(* CoDeSys 2.3.9.41 project: AVO_M.pro *)
(* Libraries: STANDARD.LIB 4.10.05 11:14:46, IECSFC.LIB 13.4.06 15:51:28, SYSLIBTIME.LIB 20.2.06 13:31:16, SYSTASKINFO.LIB 20.2.06 13:31:38, ANALYZATION.LIB 5.10.99 09:05:06, SYSLIBCALLBACK.LIB 20.2.06 13:31:08, Util.lib 18.5.10 15:14:28 *)

(* PLC configuration (modules and I/O channels)
Fast discrete inputs [I_SIMPLE_INPUT] node 0, in %IB0 out %QB0 {Filtrationtime = 10}
  AT %IX0.0 [BitInput] Discrete input 1
  AT %IX0.1 [BitInput] Discrete input 2
  AT %IX0.2 [BitInput] Discrete input 3
  AT %IX0.3 [BitInput] Discrete input 4
Discrete inputs [ID130] node 1, in %IB1 out %QB1 {Filtrationtime_GeneralINP = 10; Visibility = No; PinCount = 12}
  AT %IB1.0 [ByteInput] 8 discrete inputs
  AT %IB1.1 [ByteInput] 4 discrete inputs
Discrete outputs [ID131] node 2, in %IB2 out %QB2 {SafeValueByte = 0; SafeValueByteM = 0; Visibility = No; PinCount = 12}
  AT %QB2.0 [ByteOutput] 8 discrete outputs
  AT %QB2.1 [ByteOutput] 4 discrete outputs
Fast analog inputs [ID125] node 3, in %IB3 out %QB3 {Flt_Comm = 50Hz 2Por}
  AT %IR3.0 [FloatInputP] AI #1 {AIN_TYPE = 4-20 mA; Peak_Filtr = 200; Flt_Ch = Avr 4; TauRC = 10; MinFV = -50; MaxFV = 150}
  AT %IR3.1 [FloatInputP] AI #2 {AIN_TYPE = 4-20 mA; Peak_Filtr = 200; Flt_Ch = Off; TauRC = 10; MinFV = -50; MaxFV = 150}
  AT %IR3.2 [FloatInputP] AI #3 {AIN_TYPE = 4-20 mA; Peak_Filtr = 200; Flt_Ch = Off; TauRC = 10; MinFV = -50; MaxFV = 150}
  AT %IR3.3 [FloatInputP] AI #4 {AIN_TYPE = 4-20 mA; Peak_Filtr = 200; Flt_Ch = Off; TauRC = 10; MinFV = -50; MaxFV = 150}
  AT %IR3.4 [FloatInputP] AI #5 {AIN_TYPE = 4-20 mA; Peak_Filtr = 200; Flt_Ch = Off; TauRC = 10; MinFV = 0; MaxFV = 1.6}
  AT %IR3.5 [FloatInputP] AI #6 {AIN_TYPE = 4-20 mA; Peak_Filtr = 200; Flt_Ch = Off; TauRC = 10; MinFV = 0; MaxFV = 1.6}
  AT %IR3.6 [FloatInputP] AI #7 {AIN_TYPE = 4-20 mA; Peak_Filtr = 200; Flt_Ch = Off; TauRC = 10; MinFV = 0; MaxFV = 20000.0}
  AT %IR3.7 [FloatInputP] AI #8 {AIN_TYPE = 4-20 mA; Peak_Filtr = 200; Flt_Ch = Off; TauRC = 10; MinFV = 0; MaxFV = 20000.0}
  AT %IW3.8 [WordInput] AI read time (10ms)
Analog outputs [ID126] node 4, in %IB4 out %QB4
  AT %QR4.0 [FloatOutputP] AO #1 {AOUT_TYPE = 0-10V; SafeValueREAL = 0.0}
  AT %QR4.1 [FloatOutputP] AO #2 {AOUT_TYPE = 0-10V; SafeValueREAL = 0.0}
  AT %QR4.2 [FloatOutputP] AO #3 {AOUT_TYPE = 4-20 mA; SafeValueREAL = 0.0}
  AT %QR4.3 [FloatOutputP] AO #4 {AOUT_TYPE = 4-20 mA; SafeValueREAL = 0.0}
Special input [ID103] node 5, in %IB5 out %QB5 {Filtrationtime = 1000; PinCount = 1; WatchDogPeriod = 400; PollPeriod = 3000; Visibility = No}
  AT %IX5.0 [BitInput] Special input
Special output [ID104] node 6, in %IB6 out %QB6 {Visibility = No; PinCount = 1}
  AT %QX6.0 [BitOutput] Special output
Modbus [MODBUS_ID302] node 0, in %IB7.0 out %QB7.0
  RS-232 [COM2_USART] node 0, in %IB7.0.0 out %QB7.0.0 {CommunicationSpeed = 19200; Parity = EVEN; BitLength = 8 bits; StopLength = One stop bit; InterfaceType = RS232; FrameOriented = RTU; Timeout = 0; Visibility = No}
AT %QB7.1.0 [ByteOutput]
AT %QB7.2.0 [ByteOutput]
AT %QB7.3.0 [ByteOutput]
Float [Float] node 4, in %IB7.4 out %QB7.4
  AT %QD7.4.0 [FloatOutput]
2 byte [Register] node 5, in %IB7.5 out %QB7.5
  AT %QW7.5.0 [WordOutput]
Float [Float] node 6, in %IB7.6 out %QB7.6
  AT %QD7.6.0 [FloatOutput]
Float [Float] node 7, in %IB7.7 out %QB7.7
  AT %QD7.7.0 [FloatOutput]
Float [Float] node 8, in %IB7.8 out %QB7.8
  AT %QD7.8.0 [FloatOutput]
Float [Float] node 9, in %IB7.9 out %QB7.9
  AT %QD7.9.0 [FloatOutput]
Float [Float] node 10, in %IB7.10 out %QB7.10
  AT %QD7.10.0 [FloatOutput]
Float [Float] node 11, in %IB7.11 out %QB7.11
  AT %QD7.11.0 [FloatOutput]
Float [Float] node 12, in %IB7.12 out %QB7.12
  AT %QD7.12.0 [FloatOutput]
  AT %QD7.13.0 [FloatOutput]
Float [Float] node 14, in %IB7.14 out %QB7.14
  AT %QD7.14.0 [FloatOutput]
Float [Float] node 15, in %IB7.15 out %QB7.15
  AT %QD7.15.0 [FloatOutput]
Float [Float] node 16, in %IB7.16 out %QB7.16
  AT %QD7.16.0 [FloatOutput]
  AT %QD7.17.0 [FloatOutput]
RS-485-1 [COM1_USART] node 0, in %IB8.0.0 out %QB8.0.0 {CommunicationSpeed = 9600; Parity = NO PARITY CHECK; BitLength = 8 bits; StopLength = One stop bit; InterfaceType = RS485; FrameOriented = RTU; Timeout = 0; Visibility = No}
8 bits [8Bit] node 1, in %IB8.1 out %QB8.1
  AT %QB8.1.0 [ByteOutput]
8 bits [8Bit] node 2, in %IB8.2 out %QB8.2
  AT %QB8.2.0 [ByteOutput]
8 bits [8Bit] node 3, in %IB8.3 out %QB8.3
  AT %QB8.3.0 [ByteOutput]
8 bits [8Bit] node 4, in %IB8.4 out %QB8.4
  AT %QB8.4.0 [ByteOutput]
8 bits [8Bit] node 5, in %IB8.5 out %QB8.5
  AT %QB8.5.0 [ByteOutput]
8 bits [8Bit] node 6, in %IB8.6 out %QB8.6
  AT %QB8.6.0 [ByteOutput]
8 bits [8Bit] node 7, in %IB8.7 out %QB8.7
  AT %QB8.7.0 [ByteOutput]
8 bits [8Bit] node 8, in %IB8.8 out %QB8.8
  AT %QB8.8.0 [ByteOutput]
8 bits [8Bit] node 9, in %IB8.9 out %QB8.9
  AT %QB8.9.0 [ByteOutput]
8 bits [8Bit] node 10, in %IB8.10 out %QB8.10
  AT %QB8.10.0 [ByteOutput]
8 bits [8Bit] node 11, in %IB8.11 out %QB8.11
  AT %QB8.11.0 [ByteOutput]
  AT %QB8.12.0 [ByteOutput]
8 bits [8Bit] node 13, in %IB8.13 out %QB8.13
  AT %QB8.13.0 [ByteOutput]
8 bits [8Bit] node 14, in %IB8.14 out %QB8.14
  AT %QB8.14.0 [ByteOutput]
8 bits [8Bit] node 15, in %IB8.15 out %QB8.15
  AT %QB8.15.0 [ByteOutput]
8 bits [8Bit] node 16, in %IB8.16 out %QB8.16
  AT %QB8.16.0 [ByteOutput]
8 bits [8Bit] node 17, in %IB8.17 out %QB8.17
  AT %QB8.17.0 [ByteOutput]
8 bits [8Bit] node 18, in %IB8.18 out %QB8.18
  AT %QB8.18.0 [ByteOutput]
8 bits [8Bit] node 19, in %IB8.19 out %QB8.19
  AT %QB8.19.0 [ByteOutput]
8 bits [8Bit] node 20, in %IB8.20 out %QB8.20
  AT %QB8.20.0 [ByteOutput]
*)

(* Global variable list: Global_Variables *)
VAR_GLOBAL RETAIN
(*уставки*)
	Tnorm AT %QD7.6.0:REAL:=15;
	Tust AT %QD7.7.0:REAL:=38;
	Tmax AT %QD7.8.0:REAL:=60;
	Ti AT %QD7.12.0:REAL:=40;
	Kp AT %QD7.13.0:REAL:=0.4;
	tau_vent AT %QW7.5.0:WORD:=10;(*от 300 до 500с*)
END_VAR

VAR_GLOBAL
(*аналоговые входы*)
	t_sec AT %IR3.0:REAL;
	t_in AT %IR3.1:REAL;
	t_out AT %IR3.2:REAL;
	t_air AT %IR3.3:REAL;
	p_in AT %IR3.4:REAL;
	p_out AT %IR3.5:REAL;

(*аналоговые выходы*)
	vent1 AT %QR4.0:REAL:=0;
	vent2 AT %QR4.1:REAL:=0;

(*дискретные входы*)
	vent_kf_overheat AT %IX1.0.0:BOOL:=0; (*0 - авария, 1 - норм*)
	ten_overheat AT %IX1.0.1:BOOL:=0; (*0 - авария, 1 - норм*)
	vent1_crash AT %IX1.0.3:BOOL:=0; (*0 - авария, 1 - норм*)
	vent2_crash AT %IX1.0.4:BOOL:=0; (*0 - авария, 1 - норм*)

	qf1 AT %IX1.0.5:BOOL:=1;
	qf2 AT %IX1.0.6:BOOL:=1;
	qf5 AT %IX1.0.7:BOOL:=1;

(*дискретне выходы*)
	vent_kf AT %QX2.0.0:BOOL:=0;
	ten AT %QX2.0.1:BOOL:=0;

	t_out_high:BOOL:=0; (*превышение Тмакс*)
	p_in_high:BOOL:=0;(*превышение p_in 1,0 МПа*)
	ready:BOOL:=1;
	err:BOOL:=0;

	err_do AT %QX2.0.2:BOOL:=1; (*общая неисправность*)
	ohlad_do AT %QX2.0.3:BOOL:=1;
	norma_do AT %QX2.0.4:BOOL:=1;
	t_out_high_do AT %QX2.0.5:BOOL:=1;
	nagrev_do AT %QX2.0.6:BOOL:=1;
	ready_do AT %QX2.0.7:BOOL:=1;

(*переменные для панели*)
	nagrev AT %QX7.3.0.0:BOOL:=0;(*0-выкл,1-вкл*)
	ohlad AT %QX7.3.0.1:BOOL:=0;(*0-выкл,1-вкл*)
	norma AT %QX7.3.0.2:BOOL:=0;(*0-не норма,1-норма*)
	reg_manu AT %QX7.3.0.3:BOOL:=0;(*0-выкл,1-вкл*)

	vent1_vkl AT %QX7.2.0.0:BOOL:=TRUE;(*0-выкл,1-вкл*)
	vent2_vkl AT %QX7.2.0.1:BOOL:=TRUE;(*0-выкл,1-вкл*)

	Nust AT %QD7.11.0:REAL:=0;(*задание*)

	t_sec_pan AT %QD7.4.0:REAL;
	t_in_pan AT %QD7.9.0:REAL;
	t_out_pan AT %QD7.10.0:REAL;
	t_air_pan AT %QD7.14.0:REAL;
	p_in_pan AT %QD7.15.0:REAL;
	p_out_pan AT %QD7.16.0:REAL;

	err_pan AT %QX7.1.0.7:BOOL:=0;
	vent_kf_overheat_pan AT %QX7.1.0.2:BOOL:=0;
	ten_overheat_pan AT %QX7.1.0.3:BOOL:=0;
	t_out_high_pan AT %QX7.1.0.4:BOOL:=0;
	vent1_crash_pan AT %QX7.1.0.5:BOOL:=0;
	vent2_crash_pan AT %QX7.1.0.6:BOOL:=0;
	qf1_pan AT %QX7.2.0.2:BOOL:=1;
	qf2_pan AT %QX7.2.0.3:BOOL:=1;
	qf5_pan AT %QX7.2.0.4:BOOL:=1;


	vent_kf_pan AT %QX7.1.0.0:BOOL:=0;
	ten_pan AT %QX7.1.0.1:BOOL:=0;

(*наверх*)
	Tust_up AT %QB8.1.0:BYTE:=30;
	Tnorm_up AT %QB8.2.0:BYTE:=80;

	inp1 AT %QB8.3.0:BYTE:=15; (*рольставни, их нет на самом деле*)

	Tmax_up AT %QB8.4.0:BYTE:=160;

	inp3 AT %QB8.5.0:BYTE;
	vent_kf_overheat_up AT %QX8.5.0.2:BOOL:=0;
	ten_overheat_up AT %QX8.5.0.4:BOOL:=0;

	inp2 AT %QB8.6.0:BYTE;
	qf1_up AT %QX8.6.0.0:BOOL:=0;
	qf2_up AT %QX8.6.0.1:BOOL:=0;
	qf5_up AT %QX8.6.0.4:BOOL:=0;

	inp5 AT %QB8.7.0:BYTE;(*зарезервирован*)

	inp4 AT %QB8.8.0:BYTE;
	vent1_crash_up AT %QX8.8.0.0:BOOL:=0;
	vent2_crash_up AT %QX8.8.0.1:BOOL:=0;

	out2 AT %QB8.9.0:BYTE;
	vent1_vkl_up AT %QX8.9.0.0:BOOL:=1;(*0-выкл,1-вкл*)
	vent2_vkl_up AT %QX8.9.0.1:BOOL:=1;(*0-выкл,1-вкл*)
	vent_kf_up AT %QX2.0.0:BOOL:=0;
	ten_up AT %QX2.0.1:BOOL:=0;

	out1 AT %QB8.10.0:BYTE;(*команды на рольставни, их нет*)

	out4 AT %QB8.11.0:BYTE;
	err_up AT %QX8.11.0.0:BOOL:=1; (*0 - есть, 1 - нет*)
	ohlad_up AT %QX8.11.0.1:BOOL:=1; (*0 - есть, 1 - нет*)
	norma_up AT %QX8.11.0.2:BOOL:=1; (*0 - норма, 1 - не норма*)
	t_out_high_up AT %QX8.11.0.3:BOOL:=1; (*0 - есть, 1 - нет*)
	nagrev_up AT %QX8.11.0.4:BOOL:=0; (*0 - есть, 1 - нет*)
	ready_up AT %QX8.11.0.5:BOOL:=0; (*0 - есть, 1 - нет*)

	out3 AT %QB8.12.0:BYTE;
	sys_vkl AT %QX8.12.0.7:BOOL:=0;(*система включена, пока не используется*)

	t_out_up AT %QB8.13.0:BYTE:=90;(*по умолчанию 22*)

	out5 AT %QB8.14.0:BYTE:=0; (*номер режима охлаждения итд*)
	reg_manu_up AT %QX8.14.0.4:BOOL:=0;(*0-авт,1 - ручн*)

	t_sec_up AT %QB8.15.0:BYTE:=80;(*по умолчанию 14*)
	t_in_up AT %QB8.16.0:BYTE:=94;(*по умолчанию 25,2*)
	t_air_up AT %QB8.17.0:BYTE:=100;(*по умолчанию 30*)
	Nust_up AT %QB8.18.0:BYTE:=88;(*по умолчанию 35.2*)
	p_out_up AT %QB8.19.0:BYTE:=125;(*по умолчанию 0,001*)
	p_in_up AT %QB8.20.0:BYTE:=250;(*по умолчанию 0,002*)
END_VAR

(* POU PLC_PRG, ST *)
PROGRAM PLC_PRG
VAR
END_VAR
IF t_sec<Tnorm THEN
	nagrev:=TRUE;
ELSIF vent_kf=FALSE THEN
	nagrev:=FALSE;
END_IF

IF t_sec>=Tnorm-10 THEN
	norma:=TRUE;
ELSE
	norma:=FALSE;
END_IF

IF t_out>=Tust AND p_in>=0.2 AND norma THEN
	ohlad:=TRUE;
END_IF

IF p_in<0.2 THEN
	ohlad:=FALSE;
END_IF

IF nagrev THEN
	Tsec();
END_IF

IF ohlad THEN
	Tout();
END_IF

(*ручное регулирование*)
IF reg_manu THEN
	ohlad:=FALSE;
ELSIF NOT ohlad THEN
	Nust:=0;
END_IF

(*сигналы на вентиляторы*)
vent1:=Nust*BOOL_TO_REAL(vent1_vkl)/10;
vent2:=Nust*BOOL_TO_REAL(vent2_vkl)/10;

(*ошибки*)
errors();

(*передача параметров на панель и на САУ*)
pan();
upperlvl();
END_PROGRAM

(* POU Tsec, ST *)
PROGRAM Tsec
VAR
	delay:TOF;
	tmr:BOOL:=TRUE;
	t: TIME := T#5s;
END_VAR
t:=WORD_TO_TIME(tau_vent*1000);
IF t_sec<Tnorm-5 THEN
	vent_kf:=TRUE;
	ten:=TRUE AND NOT vent_kf_overheat;
	tmr:=TRUE;
END_IF;
IF t_sec>=Tnorm THEN
	delay(IN:=tmr,PT:=t);
	ten:=FALSE;
	tmr:=FALSE;
	vent_kf:=delay.Q;
END_IF;
END_PROGRAM

(* POU Tout, ST *)
PROGRAM Tout
VAR
	reg:PID;
	Td:REAL:=0;
END_VAR
reg(
	ACTUAL:=  t_out,
	SET_POINT:= Tust,
	KP:= -Kp,
	TN:= Ti,
	TV:= Td,
	Y_MANUAL:= Nust,
	Y_OFFSET:= 0,
	Y_MIN:= 0,
	Y_MAX:= 100,
	MANUAL:= reg_manu,
	RESET:= ,
	Y=> Nust,
	LIMITS_ACTIVE=> , 
	OVERFLOW=> );
END_PROGRAM

(* POU errors, ST *)
PROGRAM errors
VAR
END_VAR
t_out_high:=t_out>Tmax;
p_in_high:=p_in>1;

err:=NOT vent_kf_overheat OR NOT  ten_overheat OR NOT vent1_crash OR NOT vent2_crash OR t_out_high OR p_in_high OR NOT qf1 OR NOT qf2 OR NOT qf5;
ready:=NOT err;

IF NOT vent_kf_overheat THEN
ten:=FALSE;
END_IF

IF NOT vent1_crash THEN
vent1_vkl:=FALSE;
END_IF

IF NOT vent2_crash THEN
vent2_vkl:=FALSE;
END_IF
END_PROGRAM

(* POU pan, ST *)
PROGRAM pan
VAR
END_VAR
t_sec_pan:=t_sec;
t_in_pan:=t_in;
t_out_pan:=t_out;
t_air_pan:=t_air;
p_in_pan:=p_in;
p_out_pan:=p_out;

vent_kf_overheat_pan:=vent_kf_overheat;
ten_overheat_pan:=ten_overheat;
t_out_high_pan:=t_out_high;
vent1_crash_pan:=vent1_crash;
vent2_crash_pan:=vent2_crash;

vent_kf_pan:=vent_kf;
ten_pan:=ten;
END_PROGRAM

(* POU upperlvl, ST *)
PROGRAM upperlvl
VAR
END_VAR
Tnorm_up:=REAL_TO_BYTE(Tnorm*2);
Tust_up:=REAL_TO_BYTE(Tust*2);
Tmax_up:=REAL_TO_BYTE(Tmax*2);

(*inp3*)
vent_kf_overheat_up:=NOT vent_kf_overheat;
ten_overheat_up:=NOT ten_overheat;

(*inp2*)
qf1_up:=NOT qf1;
qf2_up:=NOT qf2;
qf5_up:=NOT qf5;

(*inp4*)
vent1_crash_up:=NOT vent1_crash;
vent2_crash_up:=NOT vent2_crash;

(*out2*)
vent1_vkl_up:=NOT vent1_vkl;
vent2_vkl_up:=NOT vent2_vkl;
vent_kf_up:=vent_kf;
ten_up:=ten;

(*out4*)
err_up:=NOT err;
ohlad_up:=NOT ohlad;
norma_up:=NOT norma;
t_out_high_up:=NOT t_out_high;
nagrev_up:=NOT nagrev;
ready_up:=NOT ready;

(*out5*)
reg_manu_up:=reg_manu;

t_out_up:=REAL_TO_BYTE((t_out+50)/0.8);
t_in_up:=REAL_TO_BYTE((t_in+50)/0.8);
t_air_up:=REAL_TO_BYTE((t_air+50)/0.8);
t_sec_up:=REAL_TO_BYTE((t_sec+50)/0.8);

Nust_up:=REAL_TO_BYTE(Nust/0.4);


(*дискретки*)
err_do:=NOT err;
ohlad_do:= ohlad;
norma_do:= norma;
t_out_high_do:=NOT t_out_high;
nagrev_do:= nagrev;
ready_do:= ready;
END_PROGRAM
